TYPE ST_FB_MGMT_Zustand :
STRUCT

	Betrieb_Anford			: BOOL;
	Betrieb_Soll			: BOOL;
	Betrieb					: BOOL;

	Regelung_Modus				: SINT;
	Regelung_Sollw_Widerspruch	: BOOL;
	Regelung_Sollw_Anford		: REAL;

(*Heizung*)

	Regelung_Sollw_BHKW_MBZ     : REAL;
 	Regelung_Sollw_BHKW_WBZ     : REAL;
	Regelung_Sollw_PTW1 		: REAL;
	Regelung_Sollw_BWT 		    : REAL;
	Regelung_Sollw_WP_gruennetz   : REAL;

(*Kuehlung*)
	Regelung_Sollw_blaunetz_Kuehlung 				: REAL;
	Regelung_Sollw_gruennetz_Kuehlung    : REAL;
	Regelung_Sollw_Kuehlung_KKKW            		: REAL;
	Regelung_Sollw_WP_945							:REAL;

(*Verknüpfung mit Netze*)

	Heisswasser_3xx_Zustand_Regelung_Sollw      : REAL;
	Warmwasser_2xx_Zustand_Regelung_Sollw		: REAL;
	Warmwasser_2xx_Zustand_Regelung_Sollw_Max   : REAL;
	Kaltwasser_1xx_Zustand_Regelung_Sollw 		: REAL;


	Regelung_Stellw				: REAL;
	Regelung_Istw				: REAL;

	Temp_Max				: REAL;
	Temp_Oben				: REAL;
	Temp_Min				: REAL;
	Temp_Unten				: REAL;

	Temp_KRITIKAL_OBEN_TEMP_Heissnetz  : REAL;
	Temp_KRITIKAL_UNTEN_TEMP_Heissnetz  : REAL;
	Temp_Oben_Heissnetz     : REAL;
    Temp_Unten_Heissnetz    : REAL;
	Temp_KRITIKAL_OBEN_TEMP_Warmnetz   : REAL;
	Temp_KRITIKAL_UNTEN_TEMP_Warmnetz   : REAL;
	Temp_Oben_Warmnetz      : REAL;
    Temp_Unten_Warmnetz     : REAL;
	Temp_KRITIKAL_OBEN_TEMP_Kaltnetz   : REAL;
	Temp_KRITIKAL_UNTEN_TEMP_Kaltnetz   : REAL;
	Temp_Oben_Kaltnetz      : REAL;
    Temp_Unten_Kaltnetz     : REAL;

    Temp_Hysterese_BHKW_A   : REAL;
	Temp_Hysterese_BHKW_B   : REAL;
	Temp_Hysterese_BWT		: REAL;

	Temp_Speicher795    : REAL;

	Freigabe				: BOOL;
	Freigabe_Deakt			: BOOL;
	Freigabe_Code			: WORD;
	Stoerung				: BOOL;
	Stoerung_Code			: WORD;

	Warnung					: BOOL;
	Warnung_Code			: WORD;

	Status					: SINT;
	Status_Vorl				: BOOL;
	Status_Nachl			: BOOL;

	BHKW921_Stoerung        : BOOL;
	BHKW922_Stoerung        : BOOL;

	Quittierung				: BOOL;

	Leistung			: BOOL;




END_STRUCT
END_TYPE

(* stored: Version 1.1.0.1, ProductVersion 3.1.4024.9
   DUT ST_FB_MGMT_Zustand: Id {8f5cdabd-b542-42eb-92f5-b237b10517a2} *)
